FUNCTION_BLOCK FB_BOX_DETECTOR (* Template for a Basic Function Block Type *)
  (* Standard: 61499-2 *)
  (* Version 1.0, 2022-10-13, AK123957 *)
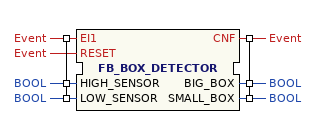
  EVENT_INPUT
    EI1 WITH HIGH_SENSOR, LOW_SENSOR; (* Sensor Data Event *)
    RESET; (* Reset Event *)
  END_EVENT
  EVENT_OUTPUT
    CNF WITH BIG_BOX, SMALL_BOX; (* Execution Confirmation *)
  END_EVENT
  VAR_INPUT
    HIGH_SENSOR : BOOL; (* Input from High Sensor *)
    LOW_SENSOR : BOOL; (* Input from Low Sensor *)
  END_VAR
  VAR_OUTPUT
    BIG_BOX : BOOL; (* True if a Big Box is Detected *)
    SMALL_BOX : BOOL; (* True if a Small Box is Detected *)
  END_VAR
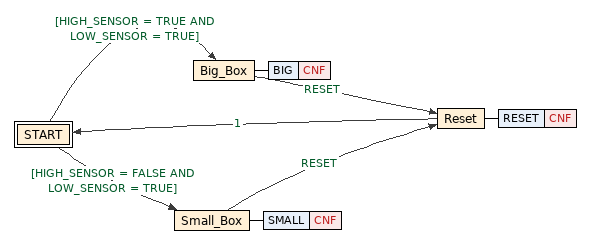
  EC_STATES
    START; (* Initial State *)
    Big_Box : BIG -> CNF;
    Small_Box : SMALL -> CNF;
    Reset : RESET -> CNF;
  END_STATES
  EC_TRANSITIONS
    START TO Big_Box := [HIGH_SENSOR = TRUE AND LOW_SENSOR = TRUE];
    START TO Small_Box := [HIGH_SENSOR = FALSE AND LOW_SENSOR = TRUE];
    Big_Box TO Reset := RESET;
    Small_Box TO Reset := RESET;
    Reset TO START := 1;
  END_TRANSITIONS
  ALGORITHM BIG IN ST:
BIG_BOX := TRUE;
SMALL_BOX := FALSE;
  END_ALGORITHM
  ALGORITHM SMALL IN ST:
BIG_BOX := FALSE;
SMALL_BOX := TRUE;
  END_ALGORITHM
  ALGORITHM RESET IN ST:
BIG_BOX:= FALSE;
SMALL_BOX := FALSE;
  END_ALGORITHM
  SERVICE left interface/right interface (* Template for a Basic Function Block Type *)
    SEQUENCE Service Sequence
      left interface.();
      left interface.EI1();
      left interface.EI1();
    END_SEQUENCE
  END_SERVICE
END_FUNCTION_BLOCK
